PROGRAM MAIN
VAR
END_VAR

CraneControl();

END_PROGRAM

(* stored: Version 1.1.0.1, ProductVersion 3.1.4024.12
   POU MAIN: Id {cc385b6b-0b41-4238-ad59-b0fe09a88c3a}, SpecialFunc None *)
